//Configuration settings for Pickup and Deposit functions to the shuttle car / Vertical Conveyor
TYPE ST_CFG_PDs_Shuttle EXTENDS ST_CFG_PDs:
STRUCT
	TiltSide 		: E_CFG_Tilt := E_CFG_Tilt.Undefined;

END_STRUCT
END_TYPE

(* stored: Version 1.1.0.1, ProductVersion 3.1.4024.9
   DUT ST_CFG_PDs_Shuttle: Id {755bb07d-09d8-4b43-a9ce-9c594ce89451} *)
